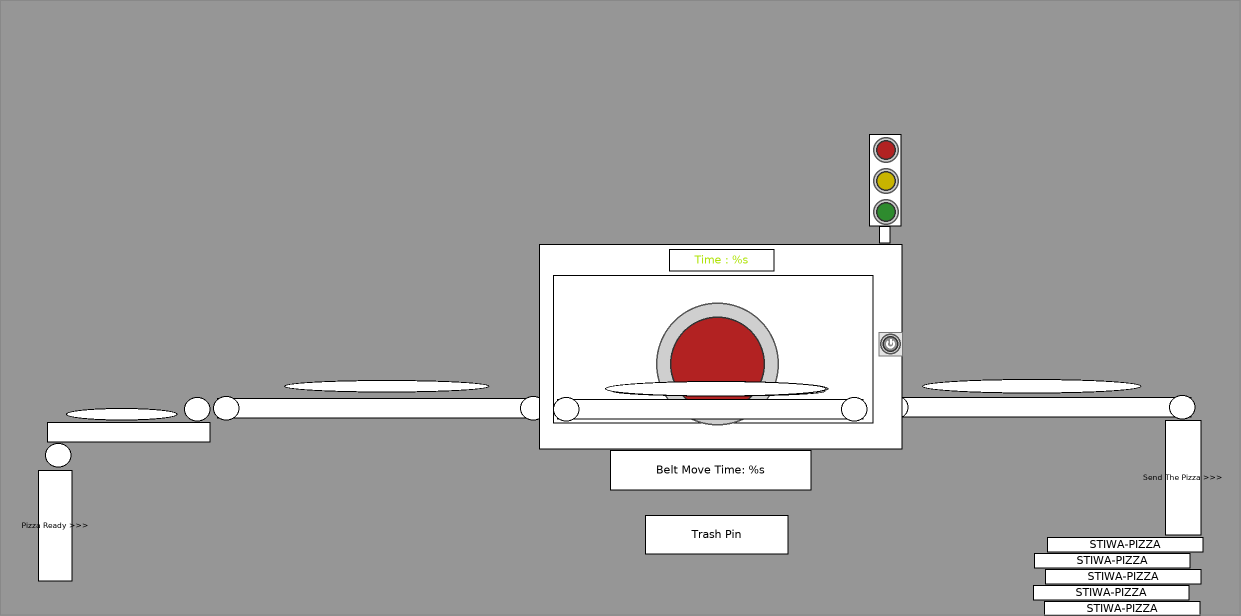
VISUALIZATION Visualization  // 1241x616
    RoundedRectangle (217,398 325x20)
    Ellipse (520,396 26x24)
    RoundedRectangle (866,397 325x20)
    Ellipse (1169,395 26x24)
    Ellipse (213,396 26x24)
    RoundedRectangle (47,422 163x20), angle 343
    Ellipse (45,443 26x24)
    Ellipse (184,397 26x24)
    Ellipse (66,408 111x12), angle 343, invisible if: NOT MAIN.MyOven.PizzaReady
    Ellipse (284,380 205x12), invisible if: NOT MAIN.MyOven.PizzaOndeck
    Ellipse (922,379 219x14), invisible if: NOT MAIN.MyOven.PizzaDone
    Rectangle (1126,459 115x36), angle 90, "Send The Pizza >>>"
        OnMouseClick: execute { MAIN.MyOven.PizzaDone:=FALSE; }
    Rectangle (0,509 111x34), angle 270, "Pizza Ready >>>"
        OnMouseClick: execute { MAIN.MyOven.PizzaReady:=TRUE; }
    Rectangle (610,450 201x40), "Belt Move Time: %s", text variable: Time_to_int(MAIN.MyOven.MoveTimer.ET)/1000
    Rectangle (1044,601 156x15), "STIWA-PIZZA"
    Rectangle (1033,585 156x15), "STIWA-PIZZA"
    Rectangle (1045,569 156x15), "STIWA-PIZZA"
    Rectangle (1034,553 156x15), "STIWA-PIZZA"
    Rectangle (1047,537 156x15), "STIWA-PIZZA"
    Rectangle (645,515 143x39), "Trash Pin"
        OnMouseClick: execute { MAIN.Step_Stat:=0; }
    Ellipse (882,395 26x24)
    Rectangle (539,244 363x205)
    RoundedRectangle (553,275 320x148)
    Lamp1 (646,279 143x170), variable: MAIN.MyOven.Power, style: Lamp-Lamp1-Red
    RoundedRectangle (557,399 306x20)
    Ellipse (841,397 26x24)
    Ellipse (553,397 26x24)
    PowerSwitch (877,332 27x24), variable: MAIN.MyOven.Power, behaviour: TOGGLE, style: Switch-PowerSwitch-Gray
    Rectangle (669,249 105x22), "Time : %s", text variable: Time_to_Int(MAIN.MyOven.OvenTimer.ET)/1000
    Ellipse (612,386 213x10), invisible if: NOT MAIN.MyOven.PizzaInOven
    Ellipse (607,381 221x15), invisible if: NOT MAIN.MyOven.PizzaIsBaked
    Ellipse (605,381 221x15), invisible if: NOT MAIN.MyOven.Burned
    RoundedRectangle (869,134 32x92)
    Lamp1 (871,197 30x30), variable: MAIN.MyOven.Power, style: Lamp-Lamp1-Green
    Lamp1 (871,135 30x30), variable: NOT MAIN.MyOven.Power, style: Lamp-Lamp1-Red
    Lamp1 (871,166 30x30), variable: MAIN.MyOven.Alarm, style: Lamp-Lamp1-Yellow
    Rectangle (879,226 11x17)
END_VISUALIZATION

(* stored: Version 1.1.0.1, ProductVersion 3.1.4024.3
   Visu Visualization: Id {2838bdb9-276b-4bcf-869a-df1a18193195} *)
